// TIA Portal project "myProject" (V18)

(* hardware
DEVICE "S7-1500/ET200MP station_1"  S7-1500 station
   slot 0: "Rail_0"  Rack  6ES7 590-1***0-0AA0
   slot 1: "PLC"  CPU 1515F-2 PN  6ES7 515-2FM02-0AB0  V2.9
      slot 3: "CPU display_1"  6ES7591-1BA00-0AA0
      slot 32768: "PROFINET interface_1"  X1
         slot 32769: "Port_1"  X1 P1
         slot 32770: "Port_2"  X1 P2
      slot 33024: "PROFINET interface_2"  X2
         slot 33025: "Port_1"  X2 P1
      slot 34817: "Virtual CP interface port_1"  Virtual CP interface port  Virtual CP interface port
*)

// ===== PLC "PLC"  CPU 1515F-2 PN =====

VAR_GLOBAL   // PLC tag table "Default tag table"
   "System_Byte" AT %MB500 : Byte;
   "FirstScan" AT %M500.0 : Bool;
   "DiagStatusUpdate" AT %M500.1 : Bool;
   "AlwaysTRUE" AT %M500.2 : Bool;
   "AlwaysFALSE" AT %M500.3 : Bool;
   "Clock_Byte" AT %MB501 : Byte;
   "Clock_10Hz" AT %M501.0 : Bool;
   "Clock_5Hz" AT %M501.1 : Bool;
   "Clock_2.5Hz" AT %M501.2 : Bool;
   "Clock_2Hz" AT %M501.3 : Bool;
   "Clock_1.25Hz" AT %M501.4 : Bool;
   "Clock_1Hz" AT %M501.5 : Bool;
   "Clock_0.625Hz" AT %M501.6 : Bool;
   "Clock_0.5Hz" AT %M501.7 : Bool;
END_VAR

DATA_BLOCK "db_Arduino Interface"   // DB2
{ S7_Optimized_Access := 'TRUE' }
VERSION : 0.1
   VAR RETAIN
      Receive : Struct
         Req : Bool;
         Disconnect : Bool;
         MB_Mode : USInt := 103;
         Connect : TCON_IP_v4;
      END_STRUCT;
   END_VAR
BEGIN
   Receive.Connect.InterfaceId := 64;
   Receive.Connect.ID := 1;
   Receive.Connect.ConnectionType := 11;
   Receive.Connect.ActiveEstablished := True;
   Receive.Connect.RemoteAddress.ADDR[1] := 192;
   Receive.Connect.RemoteAddress.ADDR[2] := 168;
   Receive.Connect.RemoteAddress.ADDR[3] := 0;
   Receive.Connect.RemoteAddress.ADDR[4] := 100;
   Receive.Connect.RemotePort := 2001;
   Receive.Connect.LocalPort := 2001;
END_DATA_BLOCK

DATA_BLOCK "db_Arduino Data"   // DB3
{ S7_Optimized_Access := 'FALSE' }
VERSION : 0.1
   VAR
      Send : Array[1..10] of Char;
   END_VAR
BEGIN
END_DATA_BLOCK

DATA_BLOCK "db_general merker"   // DB5
{ S7_Optimized_Access := 'TRUE' }
VERSION : 0.1
   VAR RETAIN
      EncoderValue : DInt;
      EncoderString : String;
      fp : Bool;
      alarm : Bool;
   END_VAR
BEGIN
END_DATA_BLOCK

DATA_BLOCK "f_db_Main Safety"   // DB5000, F_DB
{ S7_Optimized_Access := 'TRUE' }
NAME : FUSI
VERSION : 0.1
// stored: InstanceOfName fb_Main Safety
"fb_Main Safety"
BEGIN
END_DATA_BLOCK

// folder: System blocks/Program resources

DATA_BLOCK "PLC_Send_DB"   // DB4
{ S7_Optimized_Access := 'TRUE' }
AUTHOR : SIMATIC
FAMILY : MC7Plus
NAME : TC_IP_v4
VERSION : 1.0
// stored: InstanceOfName TCON_IP_v4
"TCON_IP_v4"
BEGIN
   ID := 100;
   InterfaceId := 64;
   RemotePort := 2001;
   ActiveEstablished := true;
   RemoteAddress.ADDR[1] := 192;
   RemoteAddress.ADDR[2] := 168;
   RemoteAddress.ADDR[4] := 100;
END_DATA_BLOCK

// folder: (top level)

FUNCTION_BLOCK "fb_Main Safety"   // FB5000, F_FBD
{ S7_Optimized_Access := 'TRUE' }
BEGIN
END_FUNCTION_BLOCK

ORGANIZATION_BLOCK "Main"   // OB1, LAD, ProgramCycle
TITLE = "Main Program Sweep (Cycle)"
{ S7_Optimized_Access := 'TRUE' }
VERSION : 0.1
   VAR_INPUT
      Initial_Call : Bool;   // Initial call of this OB
      Remanence : Bool;   // =True, if remanent data are available
   END_VAR
   VAR_TEMP
      done : Bool;
      busy : Bool;
      error : Bool;
      status : Word;
      index : Int;
      length : UInt;
      maxLength : Int;
   END_VAR
BEGIN

REGION Network 1 (STL)
         A     "Clock_5Hz";
         FP    "db_general merker".fp;
         JCN   x;
         L     "db_general merker".EncoderValue;
         +     1;
         T     "db_general merker".EncoderValue;
   x:    NOP   0;

         L     "db_general merker".EncoderValue;
         L     DINT#999999;
         >=I;
         JCN   y;
         L     0;
         T     "db_general merker".EncoderValue;
   y:    NOP   0;
END_REGION

REGION Network 2 (SCL): Data Management
   IF NOT "db_general merker".alarm THEN
       "db_general merker".EncoderString := DINT_TO_STRING(IN := "db_general merker".EncoderValue);
       "db_general merker".EncoderString := DELETE(IN := "db_general merker".EncoderString, L := 1, P := 1);
       #length := INT_TO_UINT(IN := LEN("db_general merker".EncoderString));
       "db_Arduino Data".Send[1] := 'e';
       Strg_TO_Chars(Strg := "db_general merker".EncoderString,
                     pChars := 1,
                     Cnt => #length,
                     Chars := "db_Arduino Data".Send);

       #maxLength := UINT_TO_INT(IN := #length);

       FOR #index := #maxLength + 2 TO 10 DO
           IF #index = #maxLength + 2 THEN
               "db_Arduino Data".Send[#index] := 'f';
           ELSE
               "db_Arduino Data".Send[#index] := ' ';
           END_IF;
       END_FOR;
   ELSE
       "db_Arduino Data".Send[1] := 'a';
       "db_Arduino Data".Send[2] := '9';
       "db_Arduino Data".Send[3] := 'f';

       FOR #index := 4 TO 10 DO
           "db_Arduino Data".Send[#index] := ' ';
       END_FOR;
   END_IF;
END_REGION

REGION Network 3 (STL): Send
   //Function
         CALL  TSEND_C , "db_Arduino Comm"
         ( REQ     := "db_Arduino Comm".REQ,
           CONT    := True,
           LEN     := 10,
           DONE    := #done,
           BUSY    := #busy,
           ERROR   := #error,
           STATUS  := #status,
           CONNECT := "PLC_Send_DB",
           DATA    := "db_Arduino Data".Send,
           ADDR    := ,
           COM_RST :=
         );

         A     "Clock_1Hz";
         =     "db_Arduino Comm".REQ;
END_REGION
END_ORGANIZATION_BLOCK